// Mitsubishi GX Works2 project: One shot ladder 1   PLC: Q03UDV

PROGRAM MAIN
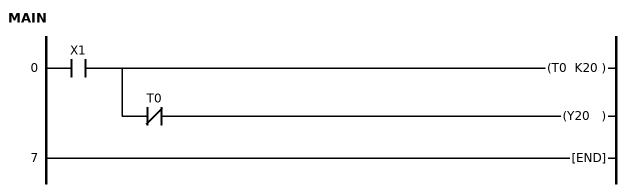
0     LD      X1
      OUT     T0 K20
      ANI     T0
      OUT     Y20
7     END
END_PROGRAM
